// TIA Portal V20 export
// export: Created 2026-08-11T18:07:18.3894618Z, ExportSetting WithDefaults, DisplayName Totally Integrated Automation Portal, DisplayVersion V20, DisplayName TIA Portal Openness, DisplayVersion V20, DisplayName TIA Portal Version Control Interface, DisplayVersion V20, DisplayName SINAMICS Startdrive Advanced, DisplayVersion V20, DisplayName SINAMICS Startdrive G130, G150, S120, S150, SINAMICS MV, G220, S200, S210, DisplayVersion V20, DisplayName SINAMICS Startdrive G110M, G120, G120C, G120D, G120P, G115D, DisplayVersion V20, DisplayName STEP 7 Professional, DisplayVersion V20, DisplayName STEP 7 Safety, DisplayVersion V20, DisplayName WinCC Basic/Comfort/Advanced, DisplayVersion V20, DisplayName WinCC Unified, DisplayVersion V20
FUNCTION_BLOCK "Program 7"   // FB15, LAD
TITLE = Proximity Sensor
{ S7_Optimized_Access := 'TRUE' }
VERSION : 0.1
// // This program simulates a hydraulic press system with safety chocks that hold the platen up. It is designed to teach how proximity sensors work as safety interlocks. The proximity sensor input (I6) verifies that the chocks are physically engaged before allowing the motors/pumps to turn off.
// 
// The proxy sits inside the press chocks and when the chocks are extended, the proxy detects the press platan and the plc knows the press is locked up and the motors can be turned off.
// 
// The chocks will not be extended unless the platan is in position, at 15000mm.
// 
// Once the chocks are extended and the platan locked up, the press is now considered to be in a safe state.
// 
// Once the user starts this worksheet/program 6,the motors will start spinning at 50% (idle), and the press platan will be on the base of the press. The user will have to click Raise, to lift the press up. Motors "under load" will spin at 100%. Then at 15000mm, the Lock button will be enabled. 
// 
// Once Lock is pressed, chocks will extend and extending will be shown until the user puts metal infront of the proximity sensor.
// 
// At this point the motor will go back to idle. And the Stop button will be enabled, for the user to stop the program. A message will then be displayed saying Press In Safe Locked Position.
// stored: AutoNumber true, IsIECCheckEnabled false, IsRetainMemResEnabled false, MemoryReserve 100, SetENOAutomatically false, UDAEnableTagReadback false
   VAR
      start { ExternalAccessible := 'False'; ExternalVisible := 'False'; ExternalWritable := 'False'} : Bool;
      motors_enable { ExternalAccessible := 'False'; ExternalVisible := 'False'; ExternalWritable := 'False'} : Bool;
      ONS : Array[0..13] of Bool;
      Machine_State : Int;
      "counter" { ExternalAccessible := 'False'; ExternalVisible := 'False'; ExternalWritable := 'False'} : Int;
      IEC : Array[0..10] of IEC_TIMER;
   END_VAR
   VAR_TEMP
      temp : Bool;
      stop_command : Bool;
      press_in_position : Bool;
      temp1 : Bool;
      temp2 : Word;
      temp3 : Word;
      random_number : DInt;
      min_value : DInt;
      max_value : DInt;
      temp4 : Real;
      temp5 : Real;
      xx : Bool;
   END_VAR
   VAR_TEMP   // added for the SCL form of the ladder/FBD networks
      _w1 : Bool;
      _w2 : Bool;
      _w3 : Bool;
      _w4 : Bool;
      _w5 : Bool;
      _w6 : Bool;
   END_VAR
BEGIN

REGION Network 1: Machine State 0 - Setup & Startup
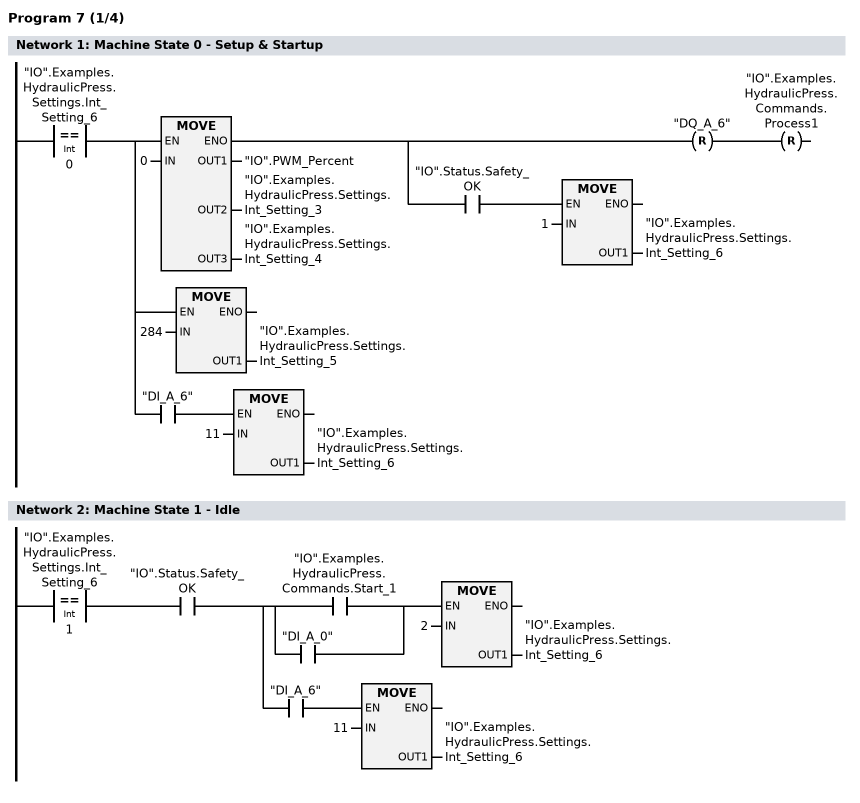
   RUNG wire#powerrail
      { S7_Templates := "SrcType := Int" } EQ_Contact(in1 := "IO".Examples.HydraulicPress.Settings.Int_Setting_6, in2 := 0)
      wire#w1
      Move(in := 0, out1 => "IO".PWM_Percent, out2 => "IO".Examples.HydraulicPress.Settings.Int_Setting_3, out3 => "IO".Examples.HydraulicPress.Settings.Int_Setting_4)
      wire#w2
      R_Coil( "DQ_A_6" )
      R_Coil( "IO".Examples.HydraulicPress.Commands.Process1 )
   END_RUNG
   RUNG wire#w2
      Contact( "IO".Status.Safety_OK )
      Move(in := 1, out1 => "IO".Examples.HydraulicPress.Settings.Int_Setting_6)
   END_RUNG
   RUNG wire#w1
      Move(in := 284, out1 => "IO".Examples.HydraulicPress.Settings.Int_Setting_5)
   END_RUNG
   RUNG wire#w1
      Contact( "DI_A_6" )
      Move(in := 11, out1 => "IO".Examples.HydraulicPress.Settings.Int_Setting_6)
   END_RUNG
   // the same network as SCL:
   #_w1 := "IO".Examples.HydraulicPress.Settings.Int_Setting_6 = 0;
   IF #_w1 THEN
       "IO".PWM_Percent := 0;
       "IO".Examples.HydraulicPress.Settings.Int_Setting_3 := 0;
       "IO".Examples.HydraulicPress.Settings.Int_Setting_4 := 0;
       "DQ_A_6" := FALSE;
       "IO".Examples.HydraulicPress.Commands.Process1 := FALSE;
   END_IF;
   IF #_w1 AND "IO".Status.Safety_OK THEN "IO".Examples.HydraulicPress.Settings.Int_Setting_6 := 1; END_IF;
   IF #_w1 THEN "IO".Examples.HydraulicPress.Settings.Int_Setting_5 := 284; END_IF;
   IF #_w1 AND "DI_A_6" THEN "IO".Examples.HydraulicPress.Settings.Int_Setting_6 := 11; END_IF;
END_REGION

REGION Network 2: Machine State 1 - Idle
   RUNG wire#powerrail
      { S7_Templates := "SrcType := Int" } EQ_Contact(in1 := "IO".Examples.HydraulicPress.Settings.Int_Setting_6, in2 := 1)
      Contact( "IO".Status.Safety_OK )
      wire#w1
      Contact( "IO".Examples.HydraulicPress.Commands.Start_1 )
      wire#w2
      Move(in := 2, out1 => "IO".Examples.HydraulicPress.Settings.Int_Setting_6)
   END_RUNG
   RUNG wire#w1
      Contact( "DI_A_0" )
   END_RUNG wire#w2
   RUNG wire#w1
      Contact( "DI_A_6" )
      Move(in := 11, out1 => "IO".Examples.HydraulicPress.Settings.Int_Setting_6)
   END_RUNG
   // the same network as SCL:
   #_w1 := ("IO".Examples.HydraulicPress.Settings.Int_Setting_6 = 1) AND "IO".Status.Safety_OK;
   IF #_w1 AND ("IO".Examples.HydraulicPress.Commands.Start_1 OR "DI_A_0") THEN
       "IO".Examples.HydraulicPress.Settings.Int_Setting_6 := 2;
   END_IF;
   IF #_w1 AND "DI_A_6" THEN "IO".Examples.HydraulicPress.Settings.Int_Setting_6 := 11; END_IF;
END_REGION

REGION Network 3: Machine State 2 - Raise
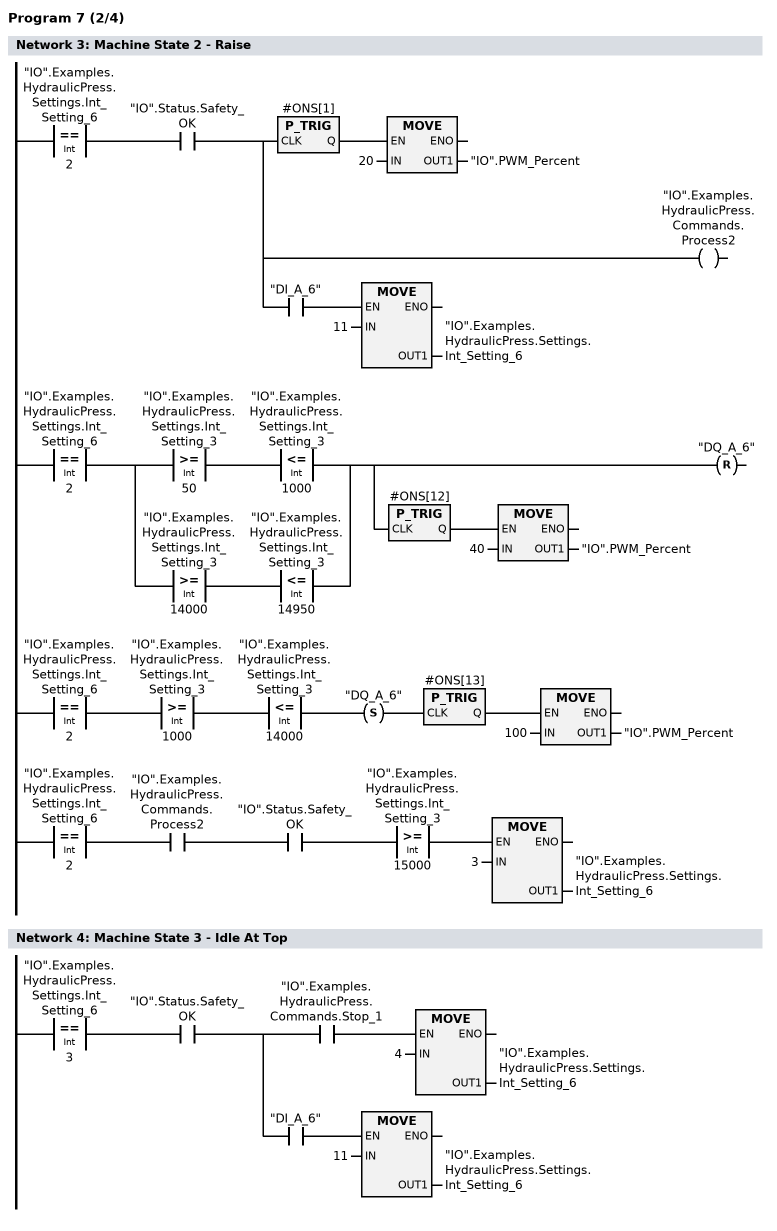
   RUNG wire#powerrail
      { S7_Templates := "SrcType := Int" } EQ_Contact(in1 := "IO".Examples.HydraulicPress.Settings.Int_Setting_6, in2 := 2)
      Contact( "IO".Status.Safety_OK )
      wire#w1
      P_Trig( #ONS[1] )
      Move(in := 20, out1 => "IO".PWM_Percent)
   END_RUNG
   RUNG wire#w1
      Coil( "IO".Examples.HydraulicPress.Commands.Process2 )
   END_RUNG
   RUNG wire#w1
      Contact( "DI_A_6" )
      Move(in := 11, out1 => "IO".Examples.HydraulicPress.Settings.Int_Setting_6)
   END_RUNG
   RUNG wire#powerrail
      { S7_Templates := "SrcType := Int" } EQ_Contact(in1 := "IO".Examples.HydraulicPress.Settings.Int_Setting_6, in2 := 2)
      wire#w2
      { S7_Templates := "SrcType := Int" } GE_Contact(in1 := "IO".Examples.HydraulicPress.Settings.Int_Setting_3, in2 := 50)
      { S7_Templates := "SrcType := Int" } LE_Contact(in1 := "IO".Examples.HydraulicPress.Settings.Int_Setting_3, in2 := 1000)
      wire#w3
      R_Coil( "DQ_A_6" )
   END_RUNG
   RUNG wire#w2
      { S7_Templates := "SrcType := Int" } GE_Contact(in1 := "IO".Examples.HydraulicPress.Settings.Int_Setting_3, in2 := 14000)
      { S7_Templates := "SrcType := Int" } LE_Contact(in1 := "IO".Examples.HydraulicPress.Settings.Int_Setting_3, in2 := 14950)
   END_RUNG wire#w3
   RUNG wire#w3
      P_Trig( #ONS[12] )
      Move(in := 40, out1 => "IO".PWM_Percent)
   END_RUNG
   RUNG wire#powerrail
      { S7_Templates := "SrcType := Int" } EQ_Contact(in1 := "IO".Examples.HydraulicPress.Settings.Int_Setting_6, in2 := 2)
      { S7_Templates := "SrcType := Int" } GE_Contact(in1 := "IO".Examples.HydraulicPress.Settings.Int_Setting_3, in2 := 1000)
      { S7_Templates := "SrcType := Int" } LE_Contact(in1 := "IO".Examples.HydraulicPress.Settings.Int_Setting_3, in2 := 14000)
      S_Coil( "DQ_A_6" )
      P_Trig( #ONS[13] )
      Move(in := 100, out1 => "IO".PWM_Percent)
   END_RUNG
   RUNG wire#powerrail
      { S7_Templates := "SrcType := Int" } EQ_Contact(in1 := "IO".Examples.HydraulicPress.Settings.Int_Setting_6, in2 := 2)
      Contact( "IO".Examples.HydraulicPress.Commands.Process2 )
      Contact( "IO".Status.Safety_OK )
      { S7_Templates := "SrcType := Int" } GE_Contact(in1 := "IO".Examples.HydraulicPress.Settings.Int_Setting_3, in2 := 15000)
      Move(in := 3, out1 => "IO".Examples.HydraulicPress.Settings.Int_Setting_6)
   END_RUNG
   // the same network as SCL:
   #_w1 := ("IO".Examples.HydraulicPress.Settings.Int_Setting_6 = 2) AND "IO".Status.Safety_OK;
   #_w2 := #_w1 AND NOT #ONS[1];   // rising edge
   #ONS[1] := #_w1;
   IF #_w2 THEN "IO".PWM_Percent := 20; END_IF;
   "IO".Examples.HydraulicPress.Commands.Process2 := #_w1;
   IF #_w1 AND "DI_A_6" THEN "IO".Examples.HydraulicPress.Settings.Int_Setting_6 := 11; END_IF;
   #_w3 := ("IO".Examples.HydraulicPress.Settings.Int_Setting_6 = 2) AND ((("IO".Examples.HydraulicPress.Settings.Int_Setting_3 >= 50) AND ("IO".Examples.HydraulicPress.Settings.Int_Setting_3 <= 1000)) OR (("IO".Examples.HydraulicPress.Settings.Int_Setting_3 >= 14000) AND ("IO".Examples.HydraulicPress.Settings.Int_Setting_3 <= 14950)));
   IF #_w3 THEN "DQ_A_6" := FALSE; END_IF;
   #_w4 := #_w3 AND NOT #ONS[12];   // rising edge
   #ONS[12] := #_w3;
   IF #_w4 THEN "IO".PWM_Percent := 40; END_IF;
   #_w5 := ("IO".Examples.HydraulicPress.Settings.Int_Setting_6 = 2) AND ("IO".Examples.HydraulicPress.Settings.Int_Setting_3 >= 1000) AND ("IO".Examples.HydraulicPress.Settings.Int_Setting_3 <= 14000);
   IF #_w5 THEN "DQ_A_6" := TRUE; END_IF;
   #_w6 := #_w5 AND NOT #ONS[13];   // rising edge
   #ONS[13] := #_w5;
   IF #_w6 THEN "IO".PWM_Percent := 100; END_IF;
   IF ("IO".Examples.HydraulicPress.Settings.Int_Setting_6 = 2) AND "IO".Examples.HydraulicPress.Commands.Process2 AND "IO".Status.Safety_OK AND ("IO".Examples.HydraulicPress.Settings.Int_Setting_3 >= 15000) THEN
       "IO".Examples.HydraulicPress.Settings.Int_Setting_6 := 3;
   END_IF;
END_REGION

REGION Network 4: Machine State 3 - Idle At Top
   RUNG wire#powerrail
      { S7_Templates := "SrcType := Int" } EQ_Contact(in1 := "IO".Examples.HydraulicPress.Settings.Int_Setting_6, in2 := 3)
      Contact( "IO".Status.Safety_OK )
      wire#w1
      Contact( "IO".Examples.HydraulicPress.Commands.Stop_1 )
      Move(in := 4, out1 => "IO".Examples.HydraulicPress.Settings.Int_Setting_6)
   END_RUNG
   RUNG wire#w1
      Contact( "DI_A_6" )
      Move(in := 11, out1 => "IO".Examples.HydraulicPress.Settings.Int_Setting_6)
   END_RUNG
   // the same network as SCL:
   #_w1 := ("IO".Examples.HydraulicPress.Settings.Int_Setting_6 = 3) AND "IO".Status.Safety_OK;
   IF #_w1 AND "IO".Examples.HydraulicPress.Commands.Stop_1 THEN
       "IO".Examples.HydraulicPress.Settings.Int_Setting_6 := 4;
   END_IF;
   IF #_w1 AND "DI_A_6" THEN "IO".Examples.HydraulicPress.Settings.Int_Setting_6 := 11; END_IF;
END_REGION

REGION Network 5: Machine State 4 - Engaging Chocks
   // The proxy sits inside the press chocks and when the chocks are extended, the proxy detects the press platan and the plc knows the press is locked up and the motors can be turned off.
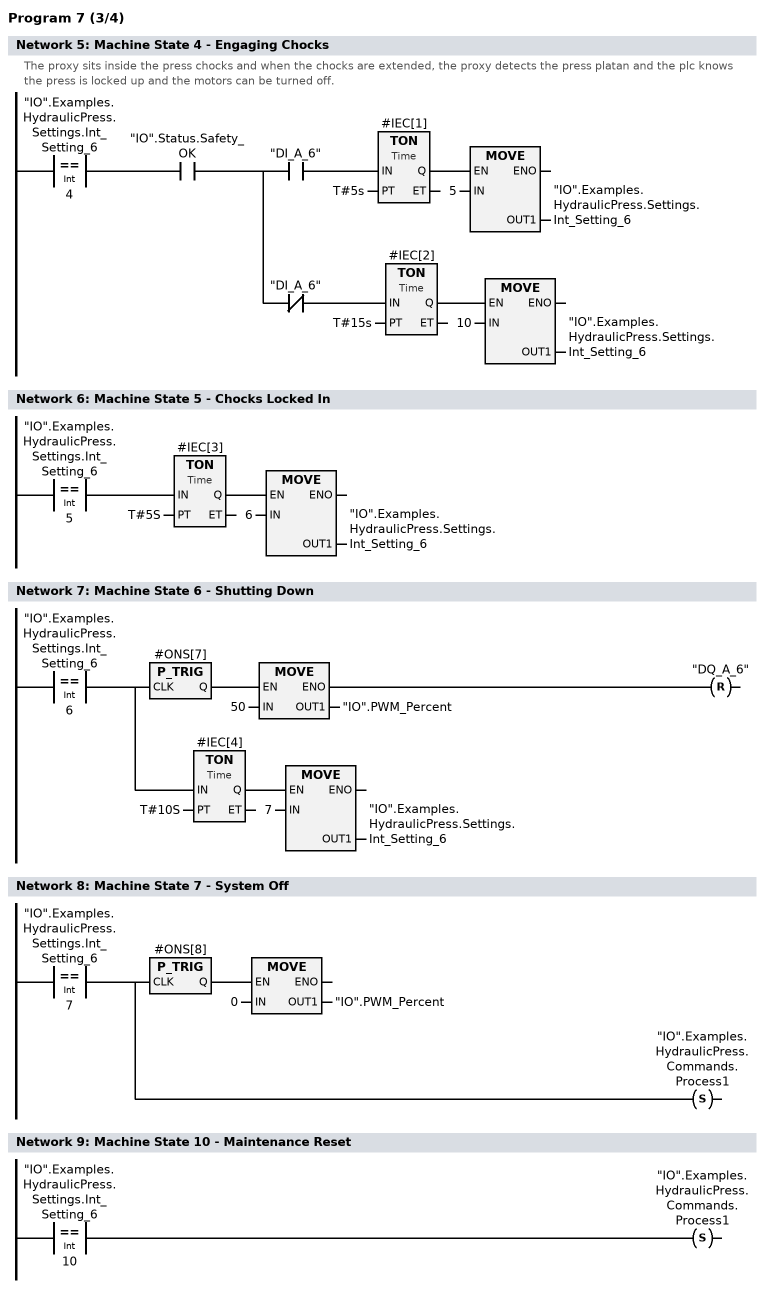
   RUNG wire#powerrail
      { S7_Templates := "SrcType := Int" } EQ_Contact(in1 := "IO".Examples.HydraulicPress.Settings.Int_Setting_6, in2 := 4)
      Contact( "IO".Status.Safety_OK )
      wire#w1
      Contact( "DI_A_6" )
      { S7_Templates := "time_type := Time" } #IEC[1].TON(pt := T#5s, et =>)
      Move(in := 5, out1 => "IO".Examples.HydraulicPress.Settings.Int_Setting_6)
   END_RUNG
   RUNG wire#w1
      I_Contact( "DI_A_6" )
      { S7_Templates := "time_type := Time" } #IEC[2].TON(pt := T#15s, et =>)
      Move(in := 10, out1 => "IO".Examples.HydraulicPress.Settings.Int_Setting_6)
   END_RUNG
   // the same network as SCL:
   #_w1 := ("IO".Examples.HydraulicPress.Settings.Int_Setting_6 = 4) AND "IO".Status.Safety_OK;
   #IEC[1].TON(IN := #_w1 AND "DI_A_6", PT := T#5s);
   IF #IEC[1].Q THEN "IO".Examples.HydraulicPress.Settings.Int_Setting_6 := 5; END_IF;
   #IEC[2].TON(IN := #_w1 AND NOT "DI_A_6", PT := T#15s);
   IF #IEC[2].Q THEN "IO".Examples.HydraulicPress.Settings.Int_Setting_6 := 10; END_IF;
END_REGION

REGION Network 6: Machine State 5 - Chocks Locked In
   RUNG wire#powerrail
      { S7_Templates := "SrcType := Int" } EQ_Contact(in1 := "IO".Examples.HydraulicPress.Settings.Int_Setting_6, in2 := 5)
      { S7_Templates := "time_type := Time" } #IEC[3].TON(pt := T#5S, et =>)
      Move(in := 6, out1 => "IO".Examples.HydraulicPress.Settings.Int_Setting_6)
   END_RUNG
   // the same network as SCL:
   #IEC[3].TON(IN := "IO".Examples.HydraulicPress.Settings.Int_Setting_6 = 5, PT := T#5S);
   IF #IEC[3].Q THEN "IO".Examples.HydraulicPress.Settings.Int_Setting_6 := 6; END_IF;
END_REGION

REGION Network 7: Machine State 6 - Shutting Down
   RUNG wire#powerrail
      { S7_Templates := "SrcType := Int" } EQ_Contact(in1 := "IO".Examples.HydraulicPress.Settings.Int_Setting_6, in2 := 6)
      wire#w1
      P_Trig( #ONS[7] )
      Move(in := 50, out1 => "IO".PWM_Percent)
      R_Coil( "DQ_A_6" )
   END_RUNG
   RUNG wire#w1
      { S7_Templates := "time_type := Time" } #IEC[4].TON(pt := T#10S, et =>)
      Move(in := 7, out1 => "IO".Examples.HydraulicPress.Settings.Int_Setting_6)
   END_RUNG
   // the same network as SCL:
   #_w1 := "IO".Examples.HydraulicPress.Settings.Int_Setting_6 = 6;
   #_w2 := #_w1 AND NOT #ONS[7];   // rising edge
   #ONS[7] := #_w1;
   IF #_w2 THEN
       "IO".PWM_Percent := 50;
       "DQ_A_6" := FALSE;
   END_IF;
   #IEC[4].TON(IN := #_w1, PT := T#10S);
   IF #IEC[4].Q THEN "IO".Examples.HydraulicPress.Settings.Int_Setting_6 := 7; END_IF;
END_REGION

REGION Network 8: Machine State 7 - System Off
   RUNG wire#powerrail
      { S7_Templates := "SrcType := Int" } EQ_Contact(in1 := "IO".Examples.HydraulicPress.Settings.Int_Setting_6, in2 := 7)
      wire#w1
      P_Trig( #ONS[8] )
      Move(in := 0, out1 => "IO".PWM_Percent)
   END_RUNG
   RUNG wire#w1
      S_Coil( "IO".Examples.HydraulicPress.Commands.Process1 )
   END_RUNG
   // the same network as SCL:
   #_w1 := "IO".Examples.HydraulicPress.Settings.Int_Setting_6 = 7;
   #_w2 := #_w1 AND NOT #ONS[8];   // rising edge
   #ONS[8] := #_w1;
   IF #_w2 THEN "IO".PWM_Percent := 0; END_IF;
   IF #_w1 THEN "IO".Examples.HydraulicPress.Commands.Process1 := TRUE; END_IF;
END_REGION

REGION Network 9: Machine State 10 - Maintenance Reset
   RUNG wire#powerrail
      { S7_Templates := "SrcType := Int" } EQ_Contact(in1 := "IO".Examples.HydraulicPress.Settings.Int_Setting_6, in2 := 10)
      S_Coil( "IO".Examples.HydraulicPress.Commands.Process1 )
   END_RUNG
   // the same network as SCL:
   IF "IO".Examples.HydraulicPress.Settings.Int_Setting_6 = 10 THEN
       "IO".Examples.HydraulicPress.Commands.Process1 := TRUE;
   END_IF;
END_REGION

REGION Network 10: Machine State 11 - Proxy Error
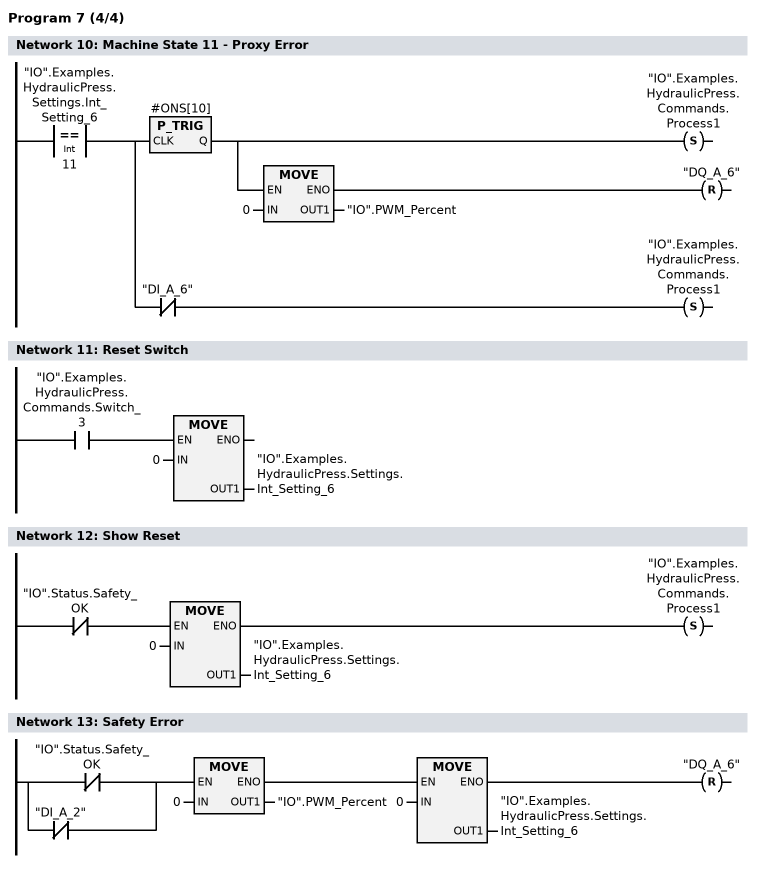
   RUNG wire#powerrail
      { S7_Templates := "SrcType := Int" } EQ_Contact(in1 := "IO".Examples.HydraulicPress.Settings.Int_Setting_6, in2 := 11)
      wire#w1
      P_Trig( #ONS[10] )
      wire#w2
      S_Coil( "IO".Examples.HydraulicPress.Commands.Process1 )
   END_RUNG
   RUNG wire#w2
      Move(in := 0, out1 => "IO".PWM_Percent)
      R_Coil( "DQ_A_6" )
   END_RUNG
   RUNG wire#w1
      I_Contact( "DI_A_6" )
      S_Coil( "IO".Examples.HydraulicPress.Commands.Process1 )
   END_RUNG
   // the same network as SCL:
   #_w1 := "IO".Examples.HydraulicPress.Settings.Int_Setting_6 = 11;
   #_w2 := #_w1 AND NOT #ONS[10];   // rising edge
   #ONS[10] := #_w1;
   IF #_w2 THEN
       "IO".Examples.HydraulicPress.Commands.Process1 := TRUE;
       "IO".PWM_Percent := 0;
       "DQ_A_6" := FALSE;
   END_IF;
   IF #_w1 AND NOT "DI_A_6" THEN "IO".Examples.HydraulicPress.Commands.Process1 := TRUE; END_IF;
END_REGION

REGION Network 11: Reset Switch
   RUNG wire#powerrail
      Contact( "IO".Examples.HydraulicPress.Commands.Switch_3 )
      Move(in := 0, out1 => "IO".Examples.HydraulicPress.Settings.Int_Setting_6)
   END_RUNG
   // the same network as SCL:
   IF "IO".Examples.HydraulicPress.Commands.Switch_3 THEN
       "IO".Examples.HydraulicPress.Settings.Int_Setting_6 := 0;
   END_IF;
END_REGION

REGION Network 12: Show Reset
   RUNG wire#powerrail
      I_Contact( "IO".Status.Safety_OK )
      Move(in := 0, out1 => "IO".Examples.HydraulicPress.Settings.Int_Setting_6)
      S_Coil( "IO".Examples.HydraulicPress.Commands.Process1 )
   END_RUNG
   // the same network as SCL:
   IF NOT "IO".Status.Safety_OK THEN
       "IO".Examples.HydraulicPress.Settings.Int_Setting_6 := 0;
       "IO".Examples.HydraulicPress.Commands.Process1 := TRUE;
   END_IF;
END_REGION

REGION Network 13: Safety Error
   RUNG wire#powerrail
      I_Contact( "IO".Status.Safety_OK )
      wire#w1
      Move(in := 0, out1 => "IO".PWM_Percent)
      Move(in := 0, out1 => "IO".Examples.HydraulicPress.Settings.Int_Setting_6)
      R_Coil( "DQ_A_6" )
   END_RUNG
   RUNG wire#powerrail
      I_Contact( "DI_A_2" )
   END_RUNG wire#w1
   // the same network as SCL:
   IF NOT "IO".Status.Safety_OK OR NOT "DI_A_2" THEN
       "IO".PWM_Percent := 0;
       "IO".Examples.HydraulicPress.Settings.Int_Setting_6 := 0;
       "DQ_A_6" := FALSE;
   END_IF;
END_REGION
END_FUNCTION_BLOCK
